TYPE Read_MainPS_Values_To_PC_Struct :
UNION
	S_MainPSValues_To_PC:S_MainPSValues_To_PC_Struct;
END_UNION
END_TYPE

(* stored: Version 1.1.0.1, ProductVersion 3.1.4024.16
   DUT Read_MainPS_Values_To_PC_Struct: Id {4cdadbf4-4ed7-4a9b-89a3-90ad03fadc07} *)
